VAR_GLOBAL
	tMotionSensorsTOF_PT		: TIME := T#5M;			//how long lamps stay lighten up after move ended
	tMotionSensorsTOF_info_PT	: TIME := T#10S;		//how long motion flags stay TRUE after move ended
	todGlobalTime				: TOD := TOD#10:0:0;
END_VAR

VAR_GLOBAL CONSTANT
	
	byStreetLampsCount			: BYTE := 10;
	byStreetLampsScenesNumber	: BYTE := 127;
	
	//Standard Brightness
	
	c_byBrightness_Alarm	: BYTE := 254;
	c_byBrightness_Motion	: BYTE := 230;
	c_byBrightness_Night	: BYTE := 180;
	c_byBrightness_Day		: BYTE := 0; 
	
	
	
END_VAR

(* stored: Version 1.1.0.1, ProductVersion 3.1.4024.5
   GVL GVL_GenSysInfo: Id {63e19513-76f4-4564-b069-1c3f57f4ab63} *)
